// TIA Portal V18 export
DATA_BLOCK "PID_correction"   // DB350
{ S7_Optimized_Access := 'TRUE' }
VERSION : 0.1
// stored: AutoNumber false, DBAccessibleFromOPCUA true, IsOnlyStoredInLoadMemory false, IsRetainMemResEnabled false, IsWriteProtectedInAS false, MemoryReserve 100
   VAR
      "Flowrate withadjustment" : Struct
         "A" : Real;
         "B" : Real;
      END_STRUCT;
      "Flowrate with adjustment_ml" : Struct
         "A" : Real;
         "B" : Real;
      END_STRUCT;
      "Manual Value" : Struct
         "A" : Real;
         "B" : Real;
      END_STRUCT;
      "Flowrate%" : Struct
         "A" : Real;
         "B" : Real;
      END_STRUCT;
      "Start manual Mode" : Struct
         "A" : Bool;
         "B" : Bool;
      END_STRUCT;
      "Start Auto Mode" : Struct
         "A" : Bool;
         "B" : Bool;
      END_STRUCT;
   END_VAR
BEGIN
END_DATA_BLOCK
